(*
Schedules jobs execution.
*)
FUNCTION_BLOCK Worker IMPLEMENTS I_Worker
VAR
	_iFirst: I_JobNode;
	_iLast: I_JobNode;	
END_VAR

(*
Defer the Job. Move it to the end of queue.
Returns:
- Ok - Success
- Err.Itf0 - iJob = 0
- Err.NoMatch = iJob.Worker <> THIS^
*)
METHOD Defer : Result
VAR_INPUT
    iJob : I_JobNode;
END_VAR
VAR
    _iPrev  : I_JobNode;
    _iNext  : I_JobNode;
    _iThis  : I_Worker := THIS^;
END_VAR
IF iJob = 0 THEN
    Defer := Err.Itf0;
    RETURN;
END_IF;

IF iJob.Worker <> _iThis THEN
    Defer := Err.NoMatch;
    RETURN;
END_IF;

_iPrev := iJob._Prev;
_iNext := iJob._Next;

IF _iPrev <> 0 THEN
    _iPrev._Next := _iNext;
ELSE
    _iFirst := _iNext;
END_IF;

IF _iNext <> 0 THEN
    _iNext._Prev := _iPrev;
ELSE
    _iLast := _iPrev;
END_IF;

iJob._Prev := _iLast;
iJob._Next := 0;

IF _iLast <> 0 THEN
    _iLast._Next := iJob;
ELSE
    _iFirst := iJob;
END_IF;

_iLast := iJob;

Defer := Ok;
END_METHOD

(*
Remove job from the queue and resets it.
Returns:
- Ok - Success
- Err.Itf0 - iJob = 0
- Err.NoMatch - iJob.Worker <> THIS^
- Err.IncArg - iJob.State = TaskState.Idle
*)
METHOD Dequeue : Result
VAR_INPUT
	iJob: I_JobNode;
END_VAR
VAR
	_iPrev: I_JobNode;
	_iNext: I_JobNode;
	_iThis: I_Worker := THIS^;
END_VAR
IF iJob = 0 THEN
	Dequeue := Err.Itf0;
    RETURN;
END_IF;

IF iJob.Worker <> _iThis THEN
    Dequeue := Err.NoMatch;
    RETURN;
END_IF;

IF iJob.State = JobState.Idle THEN
    Dequeue := Err.IncArg;
    RETURN;
END_IF;

_iPrev := iJob._Prev;
_iNext := iJob._Next;

IF _iPrev <> 0 THEN
    _iPrev._Next := _iNext;
ELSE
    _iFirst := _iNext;
END_IF;

IF _iNext <> 0 THEN
    _iNext._Prev := _iPrev;
ELSE
    _iLast := _iPrev;
END_IF;

iJob._Reset();

Dequeue := Ok;
END_METHOD

(*
Add Job to queue.
Returns:
- Ok - Success
- Err.Itf0 - iJob = 0
- Err.NoMatch - iJob.Worker <> THIS^
- Err.IncArg - iJob.State <> TaskState.Idle 
*)
METHOD Enqueue : Result
VAR_INPUT
	iJob: I_JobNode;
END_VAR
VAR
	_iThis: I_Worker := THIS^;
END_VAR
IF iJob = 0 THEN
    Enqueue := Err.Itf0;
    RETURN;
END_IF;

IF iJob.Worker <> _iThis THEN
    Enqueue := Err.NoMatch;
    RETURN;
END_IF;

IF iJob.State <> JobState.Idle THEN
    Enqueue := Err.IncArg;
    RETURN;
END_IF;

iJob._Prev := _iLast;
iJob._Next := 0;
IF _iLast <> 0 THEN
    _iLast._Next := iJob;
ELSE
    _iFirst := iJob;
END_IF;
_iLast := iJob;

Enqueue := Ok;
END_METHOD

(*
Returns first the Job in queue.
*)
PROPERTY First : I_JobNode
GET
First := _iFirst;
END_GET
END_PROPERTY

(*
Runs Worker.
*)
METHOD Run : Result
VAR_INPUT
	iJob	: I_JobNode;
END_VAR
IF iJob <> 0 THEN
	CASE iJob.State OF
		JobState.Aborted:
			Run := Ok;
		
		JobState.Completed:
			Run := Ok;	
		
		JobState.Ready:
			iJob._Run();
			Run := Ok;
	
		JobState.Error, JobState.Idle, JobState.Running:
			Run := Err.IncArg;
			
	END_CASE
ELSE
	Run := Err.Itf0;
END_IF
END_METHOD

END_FUNCTION_BLOCK

(* stored: Version 1.1.0.1
   POU Worker: Id {bdf5bac2-02d6-47f1-90f6-4bb785ea36ad}, SpecialFunc None
   Method Defer: Id {eadb621f-822e-46a7-8f87-8d6a18628a16}
   Method Dequeue: Id {1b67c59f-2d85-421b-bd6f-8786ee3aa944}
   Method Enqueue: Id {1aadc42c-8e0b-4826-bcf8-04220f1befbe}
   Property First: Id {0ef2726b-8b8c-4c46-b13c-2fec5850ea27}
   Get Get: Id {fb29ce8f-7ac5-46e9-a0ef-d876a531af6a}
   Method Run: Id {04e86e8d-8edf-4461-b2bc-3c27200c6d8d} *)
